{attribute 'qualified_only'}
{attribute 'strict'}
TYPE aE_State :
(
	Fault := 0,
	Auto := 1,
	ManRun := 2,
	ManStop := 3
);
END_TYPE

(* stored: Version 1.1.0.1, ProductVersion 3.1.4024.4
   DUT aE_State: Id {4af4cbba-ecba-476e-8816-c5249e25214a} *)
